TYPE ST_KeyValuePair : 
STRUCT
	sKey: WSTRING(127);
	sValue: STRING(255);
END_STRUCT
END_TYPE

(* stored: DUT ST_KeyValuePair: Id 337a4977-cb33-44ac-9a51-79fc217da8ce *)
